SUBAPPLICATION Uebung_222b_AX (* Standard IEC 61131-3 ALI_FB_CTUD (Adapter Version, LINT) mit Terminal-Ausgabe (PHYS) *)
  (* Standard: 61131-3; Description: Copyright (c) 2026 Meisterschulen am Ostbahnhof This program and the accompanying materials are made available under the terms of the Eclipse Public License 2.0 which is available at https://www.eclipse.org/legal/epl-2.0/ SPDX-License-Identifier: EPL-2.0 *)
  (* Version 1.1, 2026-04-21, Franz Höpfinger, Meisterschulen am Ostbahnhof, Added terminal output for counter value (PHYS) *)
  (* Version 1.0, 2026-04-21, Franz Höpfinger, Meisterschulen am Ostbahnhof, initial API and implementation (Adapter version) *)
  PACKAGE Uebungen;
  IMPORT Uebungen::const::UT::DefaultPool_Numeric::OutputNumber_N3;
  IMPORT logiBUS::io::DI::logiBUS_DI::Input_I1;
  IMPORT logiBUS::io::DI::logiBUS_DI::Input_I2;
  IMPORT logiBUS::io::DI::logiBUS_DI::Input_I3;
  IMPORT logiBUS::io::DI::logiBUS_DI::Input_I4;
  IMPORT logiBUS::io::DQ::logiBUS_DO::Output_Q1;
  IMPORT logiBUS::io::DQ::logiBUS_DO::Output_Q2;
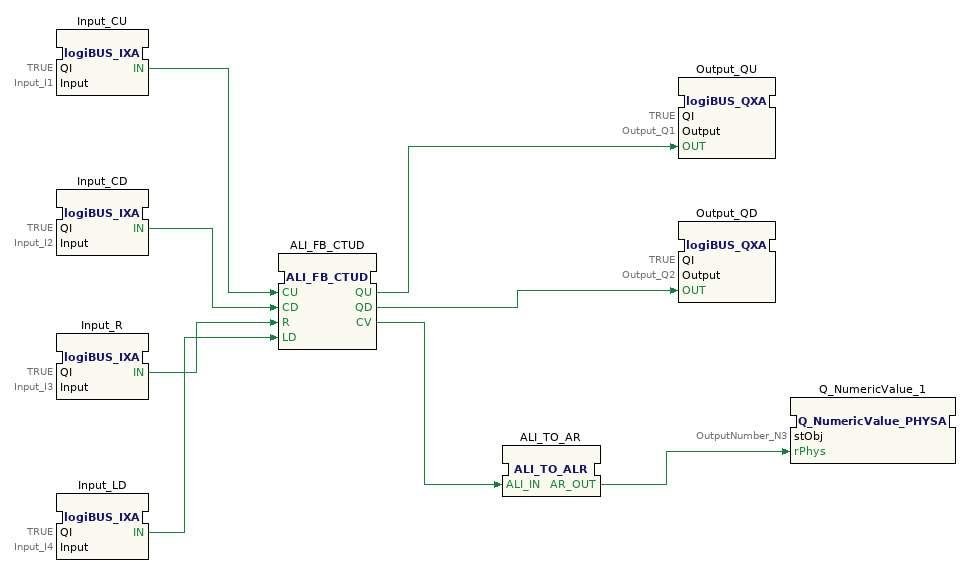
  FBS
    ALI_FB_CTUD : adapter::iec61131_3::counters::ALI_FB_CTUD;
    Input_CU : logiBUS::io::DI::logiBUS_IXA(QI := TRUE, Input := Input_I1);
    Input_CD : logiBUS::io::DI::logiBUS_IXA(QI := TRUE, Input := Input_I2);
    Input_R : logiBUS::io::DI::logiBUS_IXA(QI := TRUE, Input := Input_I3);
    Input_LD : logiBUS::io::DI::logiBUS_IXA(QI := TRUE, Input := Input_I4);
    Output_QU : logiBUS::io::DQ::logiBUS_QXA(QI := TRUE, Output := Output_Q1);
    Output_QD : logiBUS::io::DQ::logiBUS_QXA(QI := TRUE, Output := Output_Q2);
    Q_NumericValue_1 : isobus::UT::Q::Q_NumericValue_PHYSA(stObj := OutputNumber_N3);
    ALI_TO_AR : adapter::conversion::unidirectional::ALI_TO_ALR;
  END_FBS
  ADAPTER_CONNECTIONS
    Input_CU.IN TO ALI_FB_CTUD.CU;
    Input_CD.IN TO ALI_FB_CTUD.CD;
    Input_R.IN TO ALI_FB_CTUD.R;
    Input_LD.IN TO ALI_FB_CTUD.LD;
    ALI_FB_CTUD.QU TO Output_QU.OUT;
    ALI_FB_CTUD.QD TO Output_QD.OUT;
    ALI_TO_AR.AR_OUT TO Q_NumericValue_1.rPhys;
    ALI_FB_CTUD.CV TO ALI_TO_AR.ALI_IN;
  END_CONNECTIONS
END_SUBAPPLICATION
